{attribute addProperty BoxType "AX8620-0000-0027"}
{attribute addProperty Id "PSM_StatuswordAT %I*PSM_Statusword_C154CB391620WcStateAT %I*WcState_98A4DF7520.250InfoDataAT %I*InfoData_0BDED7BF144180"}
{attribute addProperty CRC "2880182750"}
{attribute addProperty SizeInBites "162"}
{attribute addProperty SizeInBytes "20.25"}
TYPE AX8620_5470AD24 :
STRUCT
	{attribute addProperty Name "PSM_Statusword"}
	PSM_Statusword : PSM_Statusword_C154CB39;
	{attribute addProperty Name "WcState"}
	WcState : WcState_98A4DF75;
	{attribute addProperty Name "InfoData"}
	InfoData : InfoData_0BDED7BF;
END_STRUCT
END_TYPE

(* stored: Version 1.2.0.0, ProductVersion 3.1.4024.9
   DUT AX8620_5470AD24: Id {d526513e-ff54-48da-8d1b-1b0d68184482} *)
